(* IEC 61131-3 sources: AXOpen/src/io/ctrl/src/AxoHwDiag/TypesStructuresAndEnums, 20 files *)

(* ---- AxoComponentState.st ---- *)
NAMESPACE AXOpen.Io
    TYPE AxoComponentState : UINT (
        Good                    :=	UINT#0, //	No problems detected.
        Disabled                :=	UINT#1, //	The hardware component is disabled.
        MaintenanceRequired     :=	UINT#2, //	Maintenance required.
        MaintenanceDemanded     :=	UINT#3, //	Maintenance demanded.
        Error                   :=	UINT#4, //	Error.
        NotAccessible           :=	UINT#5, //	Status unknown or error in higher-level hardware component.
        Unknown                 :=	UINT#6, //	Default value for components that do not return diagnostic events.
        IONotAvailable          :=	UINT#7  //	Inputs/outputs are not available.
                    ) := Unknown;
    END_TYPE
END_NAMESPACE

(* ---- AxoHwDiagComponentAvailability.st ---- *)
NAMESPACE AXOpen.Io
    TYPE AxoHwDiagComponentAvailability : UINT (
        Unknown 	            :=  UINT#255,
        Available	            :=  UINT#0,	// Hardware component is available.
        ApplicationReadyPending	:=  UINT#1,	// Application Ready Pending; no I/O access.
        LockedBySuperordinated	:=  UINT#2,	// Locked by Superordinated; no access to hardware component.
        LockedByIOController	:=  UINT#3,	// Locked by IO controller; no access to hardware component.
        LockedByIOSupervisor	:=  UINT#4	// Locked by IO supervisor; no access to hardware component.
    ) := Unknown;
    END_TYPE
END_NAMESPACE

(* ---- AxoHwDiagComponentState.st ---- *)
NAMESPACE AXOpen.Io
    TYPE AxoHwDiagComponentState : UINT (
        Good                    :=	UINT#0, //	No problems detected.
        Disabled                :=	UINT#1, //	The hardware component is disabled.
        MaintenanceRequired     :=	UINT#2, //	Maintenance required.
        MaintenanceDemanded     :=	UINT#3, //	Maintenance demanded.
        Error                   :=	UINT#4, //	Error.
        NotAccessible           :=	UINT#5, //	Status unknown or error in higher-level hardware component.
        Unknown                 :=	UINT#6, //	Default value for components that do not return diagnostic events.
        IONotAvailable          :=	UINT#7  //	Inputs/outputs are not available.
                    ) := Unknown;
    END_TYPE
END_NAMESPACE

(* ---- AxoHwDiagOperatingState.st ---- *)
NAMESPACE AXOpen.Io
    TYPE AxoHwDiagOperatingState : UINT (
        Unknown                     :=  UINT#255,
        NotSupported                :=	UINT#0,     //	Not Supported; for I/O modules OperatingState always has this value.
        StopFirmwareUpdate          :=	UINT#1,     //	STOP; firmware update.
        StopMemoryReset             :=	UINT#2,     //	STOP; memory reset.
        StopSelfStart               :=	UINT#3,     //	STOP; self start.
        Stop                        :=	UINT#4,     //	STOP.
        MemoryReset                 :=	UINT#5,     //	Memory reset.
        Startup                     :=	UINT#6,     //	STARTUP.
        Run                         :=	UINT#8,     //	RUN.
        RunRedundant                :=	UINT#9,     //	RUN-REDUNDANT.
        Hold                        :=	UINT#10,    //	HOLD.
        Defect                      :=	UINT#13,    //	DEFECT (can only be seen in diagnostic buffer entries).
        DeEnergized                 :=	UINT#15,    //	De-energized (can only be seen in diagnostic buffer entries).
        ConfigurationInRun          :=	UINT#16,    //	Configuration in Run (CiR).
        StopWithoutOutputDisable    :=	UINT#17,    //	STOP without output disable.
        RunWithOutputDisable        :=	UINT#18,    //	RUN with output disable.
        PgmTest                     :=	UINT#19,    //	PgmTest.
        PrimaryRunBackupTest        :=	UINT#20,    //	RunPgmTest (state of primary PLC when the backup PLC is in test mode).
        PrimarySyncup               :=	UINT#21,    //	RUN-SYNCUP (only primary PLC in SYNCUP system state).
        BackupSyncup                :=	UINT#22,    //	SYNCUP (only backup PLC in SYNCUP system state)
        PartnerPlcStateUnknown      :=	UINT#31,    //	State of partner PLC unknown (for example when the partner PLC is not available).
        StopSystemState             :=	UINT#33,    //	STOP system state
        StartupSystemState          :=	UINT#35,    //	STARTUP system state
        RunSoloSystemState          :=	UINT#37,    //	RUN-SOLO system state
        SyncupSystemState           :=	UINT#38,    //	SYNCUP system state
        RunRedundantSystemState     :=	UINT#40    //	RUN-REDUNDANT system state
                    ) := Unknown;
    END_TYPE
END_NAMESPACE

(* ---- AxoHwDiagReplacementState.st ---- *)
NAMESPACE AXOpen.Io
    TYPE AxoHwDiagReplacementState : UINT (
        Unknown         :=	UINT#255,
        OK              :=	UINT#0, //	The correct element exists.
        Substitute      :=	UINT#1, //	The element was replaced by a compatible element.
        Incompatible    :=	UINT#2, //	The element was replaced by an incompatible element (is reachable, but not ready for operation).
        Missing         :=	UINT#3 //	The element does not exist.
            ) := Unknown;
    END_TYPE
END_NAMESPACE

(* ---- AxoHwDiag_Component_Status.st ---- *)
NAMESPACE AXOpen.Io
    //<summary>
    // Defines the status class for hardware diagnostics.
    //</summary>
    {S7.extern=ReadWrite}
    {#ix-attr:[Container(Layout.Stack)]}
    CLASS PUBLIC AxoHwDiag_Component_Status EXTENDS AXOpen.Components.Abstractions.AxoComponent_Status
        VAR PUBLIC

        END_VAR
    END_CLASS
END_NAMESPACE

(* ---- AxoHwDiag_Config.st ---- *)
NAMESPACE AXOpen.Io
    {S7.extern=ReadWrite}
    {#ix-attr:[Container(Layout.Stack)]}
    CLASS PUBLIC AxoHwDiag_Config
        VAR PUBLIC
            {#ix-set:AttributeName = "<#Info time#>"}
<<<<<<< HEAD
            InfoTime : LTIME := LT#5S;
            {#ix-set:AttributeName = "<#Error time#>"}
            ErrorTime : LTIME := LT#10S;
            {#ix-set:AttributeName = "<#Task timeout#>"}
            TaskTimeout : LTIME := LT#50S;
=======
            InfoTime : LTIME := LT#0S;
            {#ix-set:AttributeName = "<#Error time#>"}
            ErrorTime : LTIME := LT#0S;
            {#ix-set:AttributeName = "<#Task timeout#>"}
            TaskTimeout : LTIME := LT#0S;
>>>>>>> 878
            {#ix-set:AttributeName = "<#Hardware IDs#>"}
            HWIDs : AxoHwDiag_HWIDs;
        END_VAR
    END_CLASS
END_NAMESPACE

(* ---- AxoHwDiag_Control.st ---- *)
NAMESPACE AXOpen.Io
    {S7.extern=ReadWrite}
    {#ix-attr:[Container(Layout.Stack)]}
    CLASS PUBLIC AxoHwDiag_Control
        VAR PUBLIC

        END_VAR
    END_CLASS
END_NAMESPACE

(* ---- AxoHwDiag_HWIDs.st ---- *)
NAMESPACE AXOpen.Io
   {S7.extern=ReadWrite}
	CLASS AxoHwDiag_HWIDs
      VAR PUBLIC
         {#ix-set:AttributeName = "<#Hardware ID  of the device#>"}
         HW_Device              :  UINT;
         {#ix-set:AttributeName = "<#Hardware ID of the 'in_1' submodule#>"}
         HwID_in_1            :   UINT;
         {#ix-set:AttributeName = "<#Hardware ID of the 'in_2' submodule#>"}
         HwID_in_2            :   UINT;
         {#ix-set:AttributeName = "<#Hardware ID of the 'in_3' submodule#>"}
         HwID_in_3            :   UINT;
         {#ix-set:AttributeName = "<#Hardware ID of the 'in_4' submodule#>"}
         HwID_in_4            :   UINT;
         {#ix-set:AttributeName = "<#Hardware ID of the 'in_5' submodule#>"}
         HwID_in_5            :   UINT;
         {#ix-set:AttributeName = "<#Hardware ID of the 'in_6' submodule#>"}
         HwID_in_6            :   UINT;
         {#ix-set:AttributeName = "<#Hardware ID of the 'in_7' submodule#>"}
         HwID_in_7            :   UINT;
         {#ix-set:AttributeName = "<#Hardware ID of the 'in_8' submodule#>"}
         HwID_in_8            :   UINT;
         {#ix-set:AttributeName = "<#Hardware ID of the 'in_9' submodule#>"}
         HwID_in_9            :   UINT;
         {#ix-set:AttributeName = "<#Hardware ID of the 'in_10' submodule#>"}
         HwID_in_10           :   UINT;
         {#ix-set:AttributeName = "<#Hardware ID of the 'in_11' submodule#>"}
         HwID_in_11           :   UINT;
         {#ix-set:AttributeName = "<#Hardware ID of the 'in_12' submodule#>"}
         HwID_in_12           :   UINT;
         {#ix-set:AttributeName = "<#Hardware ID of the 'in_13' submodule#>"}
         HwID_in_13           :   UINT;
         {#ix-set:AttributeName = "<#Hardware ID of the 'in_14' submodule#>"}
         HwID_in_14           :   UINT;
         {#ix-set:AttributeName = "<#Hardware ID of the 'in_15' submodule#>"}
         HwID_in_15           :   UINT;
         {#ix-set:AttributeName = "<#Hardware ID of the 'in_16' submodule#>"}
         HwID_in_16           :   UINT;
         {#ix-set:AttributeName = "<#Hardware ID of the 'in_17' submodule#>"}
         HwID_in_17           :   UINT;
         {#ix-set:AttributeName = "<#Hardware ID of the 'in_18' submodule#>"}
         HwID_in_18           :   UINT;
         {#ix-set:AttributeName = "<#Hardware ID of the 'in_19' submodule#>"}
         HwID_in_19           :   UINT;
         {#ix-set:AttributeName = "<#Hardware ID of the 'in_20' submodule#>"}
         HwID_in_20           :   UINT;
         {#ix-set:AttributeName = "<#Hardware ID of the 'out_1' submodule#>"}
         HwID_out_1           :   UINT;
         {#ix-set:AttributeName = "<#Hardware ID of the 'out_2' submodule#>"}
         HwID_out_2           :   UINT;
         {#ix-set:AttributeName = "<#Hardware ID of the 'out_3' submodule#>"}
         HwID_out_3           :   UINT;
         {#ix-set:AttributeName = "<#Hardware ID of the 'out_4' submodule#>"}
         HwID_out_4           :   UINT;
         {#ix-set:AttributeName = "<#Hardware ID of the 'out_5' submodule#>"}
         HwID_out_5           :   UINT;
         {#ix-set:AttributeName = "<#Hardware ID of the 'out_6' submodule#>"}
         HwID_out_6           :   UINT;
         {#ix-set:AttributeName = "<#Hardware ID of the 'out_7' submodule#>"}
         HwID_out_7           :   UINT;
         {#ix-set:AttributeName = "<#Hardware ID of the 'out_8' submodule#>"}
         HwID_out_8           :   UINT;
         {#ix-set:AttributeName = "<#Hardware ID of the 'out_9' submodule#>"}
         HwID_out_9           :   UINT;
         {#ix-set:AttributeName = "<#Hardware ID of the 'out_10' submodule#>"}
         HwID_out_10          :   UINT;
         {#ix-set:AttributeName = "<#Hardware ID of the 'out_11' submodule#>"}
         HwID_out_11          :   UINT;
         {#ix-set:AttributeName = "<#Hardware ID of the 'out_12' submodule#>"}
         HwID_out_12          :   UINT;
         {#ix-set:AttributeName = "<#Hardware ID of the 'out_13' submodule#>"}
         HwID_out_13          :   UINT;
         {#ix-set:AttributeName = "<#Hardware ID of the 'out_14' submodule#>"}
         HwID_out_14          :   UINT;
         {#ix-set:AttributeName = "<#Hardware ID of the 'out_15' submodule#>"}
         HwID_out_15          :   UINT;
         {#ix-set:AttributeName = "<#Hardware ID of the 'out_16' submodule#>"}
         HwID_out_16          :   UINT;
         {#ix-set:AttributeName = "<#Hardware ID of the 'out_17' submodule#>"}
         HwID_out_17          :   UINT;
         {#ix-set:AttributeName = "<#Hardware ID of the 'out_18' submodule#>"}
         HwID_out_18          :   UINT;
         {#ix-set:AttributeName = "<#Hardware ID of the 'out_19' submodule#>"}
         HwID_out_19          :   UINT;
         {#ix-set:AttributeName = "<#Hardware ID of the 'out_20' submodule#>"}
         HwID_out_20          :   UINT;
      END_VAR
   END_CLASS
END_NAMESPACE

(* ---- AxoHwDiag_In.st ---- *)
NAMESPACE AXOpen.Io
    {S7.extern=ReadWrite}
    {#ix-attr:[Container(Layout.Wrap)]}
    CLASS PUBLIC AxoHwDiag_In
        VAR PUBLIC
            {#ix-set:AttributeName = "<#Status#>"}
            {#ix-attr:[ReadOnly()]}
            Status           :   AxoHwDiag_Status;
        END_VAR
    END_CLASS
END_NAMESPACE

(* ---- AxoHwDiag_Out.st ---- *)
NAMESPACE AXOpen.Io
    {S7.extern=ReadWrite}
    {#ix-attr:[Container(Layout.Wrap)]}
    CLASS PUBLIC AxoHwDiag_Out
        VAR PUBLIC
            {#ix-set:AttributeName = "<#Control#>"}
            {#ix-attr:[ReadOnly()]}
            Control           :   AxoHwDiag_Control;
        END_VAR
    END_CLASS
END_NAMESPACE

(* ---- AxoHwDiag_Status.st ---- *)
NAMESPACE AXOpen.Io
    {S7.extern=ReadWrite}
    {#ix-attr:[Container(Layout.Stack)]}
    CLASS PUBLIC AxoHwDiag_Status
        VAR PUBLIC

        END_VAR
    END_CLASS
END_NAMESPACE

(* ---- AxoHwDiagCommonDetails.st ---- *)
NAMESPACE AXOpen.Io
    {S7.extern=ReadWrite}
    CLASS AxoHwDiagCommonDetails
        VAR PUBLIC
            {#ix-attr:[Container(Layout.Stack)]}
            {#ix-set:AttributeName = "<#HardwareID#>"}
            HardwareID          :	UINT;
            {#ix-set:AttributeName = "<#State#>"}
            State    :	AxoComponentState;
            {#ix-set:AttributeName = "<#Subordinate state#>"}
            SubordinateState    :	AxoComponentState;
            {#ix-set:AttributeName = "<#GetDiagnosticsReturnCode#>"}
            GetDiagnosticsReturnCode : GetDiagnosticsReturnCode;
            {#ix-set:AttributeName = "<#Operating DiagnosticsEnabled#>"}
            DiagnosticsEnabled  :	BOOL;
            {#ix-set:AttributeName = "<#IO state#>"}
            IOState  :	AxoHwDiagIoState;
        END_VAR
    END_CLASS
END_NAMESPACE

(* ---- AxoHwDiagComponentStateDetail.st ---- *)
NAMESPACE AXOpen.Io
    {S7.extern=ReadWrite}
    CLASS AxoHwDiagComponentStateDetail
		VAR PUBLIC
            {#ix-attr:[Container(Layout.Wrap)]}
            {#ix-attr:[Group(GroupLayout.GroupBox)]}
            {#ix-set:AttributeName = "<#Hardware component state#>"}
            HardwareComponentState  :   AxoHwDiagHardwareComponentState;
            {#ix-attr:[Container(Layout.Wrap)]}
            {#ix-attr:[Group(GroupLayout.GroupBox)]}
            {#ix-set:AttributeName = "<#IO state#>"}
            IOState                 :	AxoHwDiagIOState;
        END_VAR
    END_CLASS
END_NAMESPACE

(* ---- AxoHwDiagDetails.st ---- *)
NAMESPACE AXOpen.Io
    {S7.extern=ReadWrite}
    {#ix-attr:[Container(Layout.Wrap)]}
    CLASS AxoHwDiagDetails
        VAR PUBLIC
            {#ix-attr:[Container(Layout.Stack)]}
            {#ix-attr:[Group(GroupLayout.GroupBox)]}
            {#ix-set:AttributeName = "<#PLC#>"}
            {#ix-attr:[ReadOnly()]}
            PLCSubSystemDiagnosticDetails	        :   AxoHwDiagSubSystemDetails;

            {#ix-attr:[Container(Layout.Stack)]}
            {#ix-attr:[Group(GroupLayout.GroupBox)]}
            {#ix-set:AttributeName = "<#IOSystem#>"}
            {#ix-attr:[ReadOnly()]}
            IoSystemSubSystemDiagnosticDetails	        :   AxoHwDiagSubSystemDetails;

            {#ix-attr:[Container(Layout.Stack)]}
            {#ix-attr:[Group(GroupLayout.GroupBox)]}
            {#ix-set:AttributeName = "<#Station#>"}
            {#ix-attr:[ReadOnly()]}
            StationSubSystemDiagnosticDetails	        :   AxoHwDiagSubSystemDetails;

            {#ix-attr:[Container(Layout.Stack)]}
            {#ix-attr:[Group(GroupLayout.GroupBox)]}
            {#ix-set:AttributeName = "<#Module#>"}
            {#ix-attr:[ReadOnly()]}
            ModuleSubSystemDiagnosticDetails	        :   AxoHwDiagSubSystemDetails;

            {#ix-attr:[Container(Layout.Stack)]}
            {#ix-attr:[Group(GroupLayout.GroupBox)]}
            {#ix-set:AttributeName = "<#Sub module#>"}
            {#ix-attr:[ReadOnly()]}
            SubModuleSubSystemDiagnosticDetails	        :   AxoHwDiagSubSystemDetails;

            {#ix-attr:[Container(Layout.Stack)]}
            {#ix-attr:[Group(GroupLayout.GroupBox)]}
            {#ix-set:AttributeName = "<#Details#>"}
            {#ix-attr:[ReadOnly()]}
            SystemDiagnosticDetails	                    :   AxoHwDiagSystemDetails;

        END_VAR
    END_CLASS
END_NAMESPACE

(* ---- AxoHwDiagHardwareComponentState.st ---- *)
NAMESPACE AXOpen.Io
    {S7.extern=ReadWrite}
    CLASS AxoHwDiagHardwareComponentState
	VAR PUBLIC
            {#ix-attr:[Container(Layout.Stack)]}
            NoAdditionalInformation     :	BOOL;	//  No additional information available.
            TransferNotPermitted        :	BOOL;	//  Transfer not permitted.
            DiagnosticsAvailable        :	BOOL;	//  At least one qualified diagnostics is available.
            MaintenanceRequired         :	BOOL;	//  Maintenance required for at least one channel or the component.
            MaintenanceDemanded         :	BOOL;	//  Maintenance demanded for at least one channel or the component.
            Error                       :	BOOL;	//  Error in at least one channel or the component.
            ComponentAvailability	    :   AxoHwDiagComponentAvailability;
            ReplacementState	        :   AxoHwDiagReplacementState;
        END_VAR
    END_CLASS
END_NAMESPACE

(* ---- AxoHwDiagIoState.st ---- *)
NAMESPACE AXOpen.Io
    {S7.extern=ReadWrite}
    CLASS AxoHwDiagIoState
        VAR PUBLIC
            {#ix-attr:[Container(Layout.Stack)]}
            Good                    :	BOOL;   //	No problems detected.
            Disabled                :	BOOL;   //	The hardware component is disabled.
            MaintenanceRequired     :	BOOL;   //	Maintenance required.
            MaintenanceDemanded     :	BOOL;   //	Maintenance demanded.
            Error                   :	BOOL;   //	Error.
            NotAccessible           :	BOOL;   //	Hardware component not reachable; hardware component cannot be accessed.
            DiagnosticsAvailable    :	BOOL;   //	At least one qualified diagnostics is available.
            IODataNotAvailable      :	BOOL;   //	I/O data not available.
            NetworkError            :	BOOL;   //	Network error.
            HardwareError           :	BOOL;   //	Hardware error.
        END_VAR
    END_CLASS
END_NAMESPACE

(* ---- AxoHwDiagPlcState.st ---- *)
NAMESPACE AXOpen.Io
    {S7.extern=ReadWrite}
    CLASS AxoHwDiagPlcState
        VAR PUBLIC
            {#ix-attr:[Container(Layout.Stack)]}
            ModuleDisabled              :   BOOL;   //	Submodule or module disabled.
            ConfigurationInRunActive    :   BOOL;   //	Configuration in Run (CiR) operation is active.
            InputNotAvailable           :   BOOL;   //	Input not available.
            OutputNotAvailable          :   BOOL;   //	Output not available.
            DiagnosticsBufferOverflow   :   BOOL;   //	Overflow of diagnostic buffer.
            DiagnosticsNotAvailable     :   BOOL;   //	Diagnostics not available.
            PartialDeviceFailure        :   BOOL;   //	Partial device failure (with PNIO for Shared iDevices).
        END_VAR
    END_CLASS
END_NAMESPACE

(* ---- AxoHwDiagSubSystemDetails.st ---- *)
NAMESPACE AXOpen.Io
    {S7.extern=ReadWrite}
    CLASS AxoHwDiagSubSystemDetails
        VAR PUBLIC
            {#ix-attr:[Container(Layout.Stack)]}
            {#ix-set:AttributeName = "<#HardwareID#>"}
            HardwareID          :	UINT;
            {#ix-set:AttributeName = "<#Subordinate state#>"}
            SubordinateState    :	AxoComponentState;
            {#ix-set:AttributeName = "<#GetDiagnosticsReturnCode#>"}
            GetDiagnosticsReturnCode : GetDiagnosticsReturnCode;
            {#ix-set:AttributeName = "<#Operating DiagnosticsEnabled#>"}
            DiagnosticsEnabled  :	BOOL;
            {#ix-set:AttributeName = "<#Subordinate IO state#>"}
            SubordinateIOState  :	AxoHwDiagIoState;
        END_VAR
    END_CLASS
END_NAMESPACE

(* ---- AxoHwDiagSystemDetails.st ---- *)
NAMESPACE AXOpen.Io
    {S7.extern=ReadWrite}
    CLASS AxoHwDiagSystemDetails
        VAR PUBLIC
            {#ix-attr:[Container(Layout.Stack)]}
            {#ix-set:AttributeName = "<#HardwareID#>"}
            HardwareID          :	UINT;
            {#ix-set:AttributeName = "<#GetDiagnosticsReturnCode#>"}
            GetDiagnosticsReturnCode : GetDiagnosticsReturnCode;
            {#ix-attr:[Container(Layout.Wrap)]}
            ComponentStateDetail    :	AxoHwDiagComponentStateDetail;
            {#ix-attr:[Container(Layout.Wrap)]}
            {#ix-set:AttributeName = "<#Component state#>"}
            ComponentState          :	AxoHwDiagComponentState;
            {#ix-attr:[Container(Layout.Wrap)]}
            {#ix-set:AttributeName = "<#Operating state#>"}
            OperatingState           :	AxoHwDiagOperatingState;
        END_VAR
    END_CLASS
END_NAMESPACE
